// TIA Portal V17 program export: 1 tag tables, 0 data types, 1 data blocks, 5 code blocks (in call order from the OBs), 13 instance data blocks

VAR_GLOBAL   // PLC tag table "Default tag table"
   System_Byte AT %MB1 : Byte;
   FirstScan AT %M1.0 : Bool;
   DiagStatusUpdate AT %M1.1 : Bool;
   AlwaysTRUE AT %M1.2 : Bool;
   AlwaysFALSE AT %M1.3 : Bool;
   Clock_Byte AT %MB0 : Byte;
   Clock_10Hz AT %M0.0 : Bool;
   Clock_5Hz AT %M0.1 : Bool;
   "Clock_2.5Hz" AT %M0.2 : Bool;
   Clock_2Hz AT %M0.3 : Bool;
   "Clock_1.25Hz" AT %M0.4 : Bool;
   Clock_1Hz AT %M0.5 : Bool;
   "Clock_0.625Hz" AT %M0.6 : Bool;
   "Clock_0.5Hz" AT %M0.7 : Bool;
   BMS_Connect_req AT %M2.0 : Bool;
   Send_data AT %M2.2 : Bool;
   Kinco_connect_req AT %M2.1 : Bool;
   Node_ID_1 AT %MW4 : Int;
   Node_ID_2 AT %MW6 : Int;
   Connection_Established AT %M2.3 : Bool;
   Motor_1_Select_mode AT %MB3 : Byte;
   move_data_pulse AT %M2.4 : Bool;
   motor_1_control_word AT %MW10 : Word;
   LH_pulse_out AT %M2.6 : Bool;
   RH_pulse_out AT %M2.7 : Bool;
   RH_Speed AT %MD18 : DInt;
   LH_Speed AT %MD22 : DInt;
   send_data_pulse AT %M2.5 : Bool;
   node_terminate AT %I0.0 : Bool;
   motor_1_target_rpm AT %MD12 : DInt;
   motor_1_target_pos AT %MD28 : DInt;
   motor_1_profile_speed AT %MD32 : DInt;
   Tag_1 AT %I0.2 : Bool;
   wake_node_trigger AT %I0.1 : Bool;
   Motor_2_Select_mode AT %MB8 : Byte;
   motor_2_control_word AT %MW16 : Word;
   motor_2_target_rpm AT %MD36 : DInt;
   motor_2_target_pos AT %MD40 : DInt;
   motor_2_profile_speed AT %MD44 : DInt;
END_VAR

DATA_BLOCK "kinco_Data_packet_DB"   // DB9
{ S7_Optimized_Access := 'FALSE' }
VERSION : 0.1
// stored: AutoNumber true, DBAccessibleFromOPCUA true, IsOnlyStoredInLoadMemory false, IsWriteProtectedInAS false
   VAR
      Kinco_Data_Recv : Array[0..12] of Byte;
      Kinco_Data_sending_vizu : Array[0..12] of Byte;
   END_VAR
BEGIN
END_DATA_BLOCK

ORGANIZATION_BLOCK "Main"   // OB1, LAD, ProgramCycle
TITLE = "Main Program Sweep (Cycle)"
{ S7_Optimized_Access := 'TRUE' }
VERSION : 0.1
// stored: AutoNumber true, IsIECCheckEnabled false, SetENOAutomatically false
   VAR_INPUT
      Initial_Call : Bool;   // Initial call of this OB
      Remanence : Bool;   // =True, if remanent data are available
   END_VAR
BEGIN

REGION Network 1
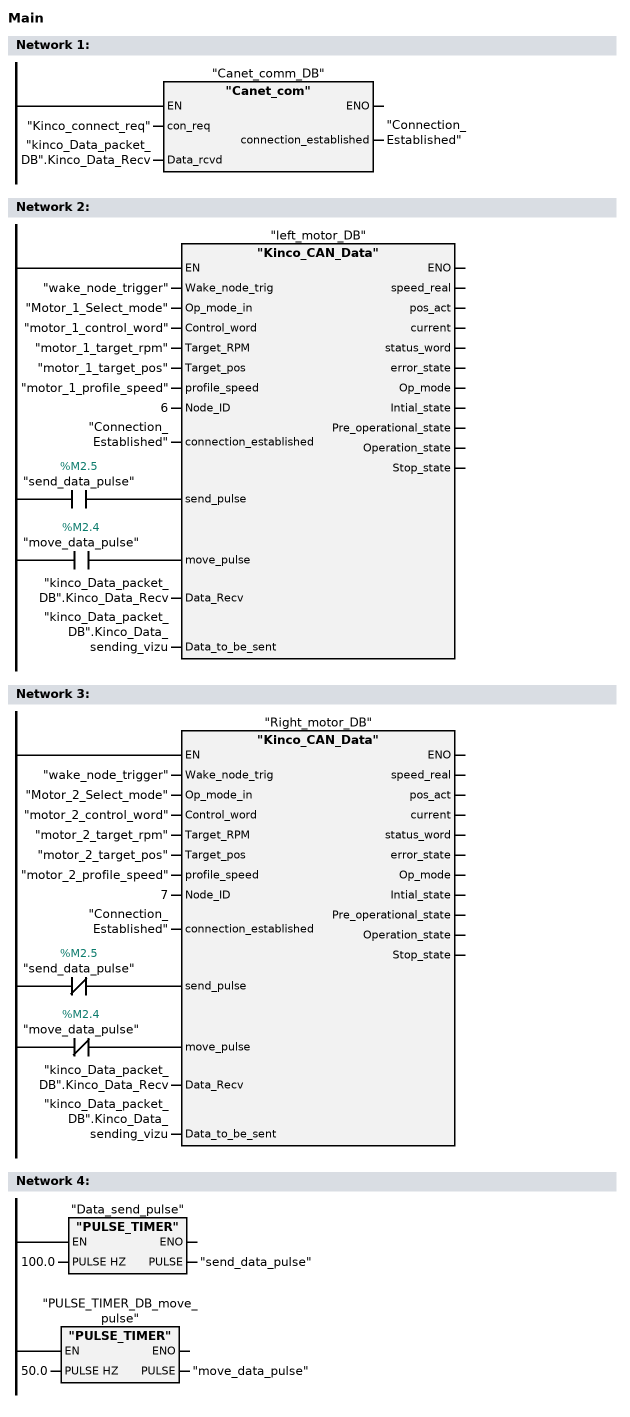
   RUNG wire#powerrail
      "Canet_comm_DB"(con_req := "Kinco_connect_req", Data_rcvd := "kinco_Data_packet_DB".Kinco_Data_Recv, connection_established => "Connection_Established")
   END_RUNG
   // the same network as SCL:
   "Canet_comm_DB"(con_req := "Kinco_connect_req",   // "Canet_com"
                   Data_rcvd := "kinco_Data_packet_DB".Kinco_Data_Recv,
                   connection_established => "Connection_Established");
END_REGION

REGION Network 2
   RUNG wire#powerrail
      "left_motor_DB"(send_pulse := wire#w1, move_pulse := wire#w2, Wake_node_trig := "wake_node_trigger", Op_mode_in := "Motor_1_Select_mode", Control_word := "motor_1_control_word", Target_RPM := "motor_1_target_rpm", Target_pos := "motor_1_target_pos", profile_speed := "motor_1_profile_speed", Node_ID := 6, connection_established := "Connection_Established", Data_Recv := "kinco_Data_packet_DB".Kinco_Data_Recv, Data_to_be_sent := "kinco_Data_packet_DB".Kinco_Data_sending_vizu, speed_real =>, pos_act =>, current =>, status_word =>, error_state =>, Op_mode =>, Intial_state =>, Pre_operational_state =>, Operation_state =>, Stop_state =>)
   END_RUNG
   RUNG wire#powerrail
      Contact( "send_data_pulse" )
   END_RUNG wire#w1
   RUNG wire#powerrail
      Contact( "move_data_pulse" )
   END_RUNG wire#w2
   // the same network as SCL:
   "left_motor_DB"(Wake_node_trig := "wake_node_trigger",   // "Kinco_CAN_Data"
                   Op_mode_in := "Motor_1_Select_mode",
                   Control_word := "motor_1_control_word",
                   Target_RPM := "motor_1_target_rpm",
                   Target_pos := "motor_1_target_pos",
                   profile_speed := "motor_1_profile_speed",
                   Node_ID := 6,
                   connection_established := "Connection_Established",
                   send_pulse := "send_data_pulse",
                   move_pulse := "move_data_pulse",
                   Data_Recv := "kinco_Data_packet_DB".Kinco_Data_Recv,
                   Data_to_be_sent := "kinco_Data_packet_DB".Kinco_Data_sending_vizu);
END_REGION

REGION Network 3
   RUNG wire#powerrail
      "Right_motor_DB"(send_pulse := wire#w1, move_pulse := wire#w2, Wake_node_trig := "wake_node_trigger", Op_mode_in := "Motor_2_Select_mode", Control_word := "motor_2_control_word", Target_RPM := "motor_2_target_rpm", Target_pos := "motor_2_target_pos", profile_speed := "motor_2_profile_speed", Node_ID := 7, connection_established := "Connection_Established", Data_Recv := "kinco_Data_packet_DB".Kinco_Data_Recv, Data_to_be_sent := "kinco_Data_packet_DB".Kinco_Data_sending_vizu, speed_real =>, pos_act =>, current =>, status_word =>, error_state =>, Op_mode =>, Intial_state =>, Pre_operational_state =>, Operation_state =>, Stop_state =>)
   END_RUNG
   RUNG wire#powerrail
      I_Contact( "send_data_pulse" )
   END_RUNG wire#w1
   RUNG wire#powerrail
      I_Contact( "move_data_pulse" )
   END_RUNG wire#w2
   // the same network as SCL:
   "Right_motor_DB"(Wake_node_trig := "wake_node_trigger",   // "Kinco_CAN_Data"
                    Op_mode_in := "Motor_2_Select_mode",
                    Control_word := "motor_2_control_word",
                    Target_RPM := "motor_2_target_rpm",
                    Target_pos := "motor_2_target_pos",
                    profile_speed := "motor_2_profile_speed",
                    Node_ID := 7,
                    connection_established := "Connection_Established",
                    send_pulse := NOT "send_data_pulse",
                    move_pulse := NOT "move_data_pulse",
                    Data_Recv := "kinco_Data_packet_DB".Kinco_Data_Recv,
                    Data_to_be_sent := "kinco_Data_packet_DB".Kinco_Data_sending_vizu);
END_REGION

REGION Network 4
   RUNG wire#powerrail
      "Data_send_pulse"("PULSE HZ" := 100.0, PULSE => "send_data_pulse")
   END_RUNG
   RUNG wire#powerrail
      "PULSE_TIMER_DB_move_pulse"("PULSE HZ" := 50.0, PULSE => "move_data_pulse")
   END_RUNG
   // the same network as SCL:
   "Data_send_pulse"("PULSE HZ" := 100.0, PULSE => "send_data_pulse");   // "PULSE_TIMER"
   "PULSE_TIMER_DB_move_pulse"("PULSE HZ" := 50.0, PULSE => "move_data_pulse");   // "PULSE_TIMER"
END_REGION
END_ORGANIZATION_BLOCK

FUNCTION_BLOCK "Canet_com"   // FB3, LAD
{ S7_Optimized_Access := 'FALSE' }
VERSION : 0.1
// stored: AutoNumber true, IsIECCheckEnabled false, SetENOAutomatically false, UDAEnableTagReadback false
   VAR_INPUT
      con_req : Bool;
   END_VAR
   VAR_OUTPUT
      connection_established : Bool;
   END_VAR
   VAR_IN_OUT
      Data_rcvd : Array[0..12] of Byte;
   END_VAR
BEGIN

REGION Network 1: Connection
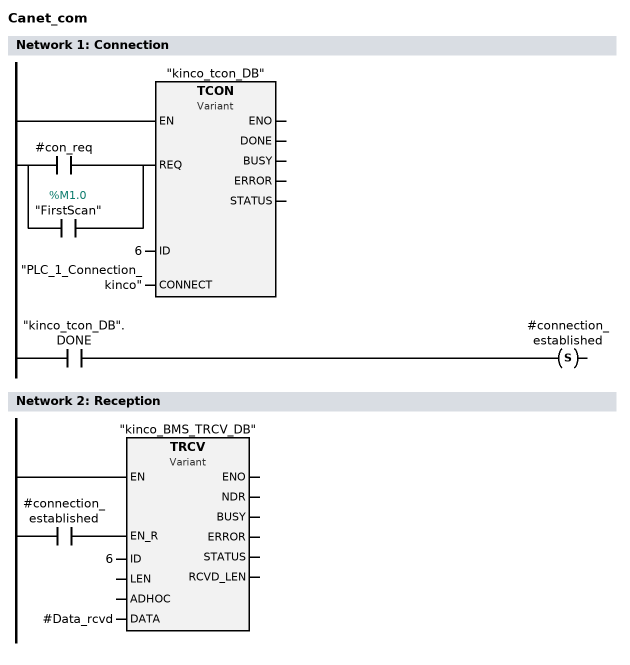
   RUNG wire#powerrail
      { S7_Templates := "[con_type := Variant, id_type := CONN_OUC]" } "kinco_tcon_DB".TCON(REQ := wire#w1, ID := 6, CONNECT := "PLC_1_Connection_kinco", DONE =>, BUSY =>, ERROR =>, STATUS =>)
   END_RUNG
   RUNG wire#powerrail
      Contact( #con_req )
   END_RUNG wire#w1
   RUNG wire#powerrail
      Contact( "FirstScan" )
   END_RUNG wire#w1
   RUNG wire#powerrail
      Contact( "kinco_tcon_DB".DONE )
      S_Coil( #connection_established )
   END_RUNG
   // the same network as SCL:
   "kinco_tcon_DB"(REQ := #con_req OR "FirstScan", ID := 6, CONNECT := "PLC_1_Connection_kinco");   // TCON
   IF "kinco_tcon_DB".DONE THEN #connection_established := TRUE; END_IF;
END_REGION

REGION Network 2: Reception
   RUNG wire#powerrail
      { S7_Templates := "[card := 1, ptr_type := Variant, value_type := UDInt, id_type := CONN_OUC]" } "kinco_BMS_TRCV_DB".TRCV(EN_R := wire#w1, ID := 6, LEN :=, ADHOC :=, DATA := #Data_rcvd, NDR =>, BUSY =>, ERROR =>, STATUS =>, RCVD_LEN =>)
   END_RUNG
   RUNG wire#powerrail
      Contact( #connection_established )
   END_RUNG wire#w1
   // the same network as SCL:
   "kinco_BMS_TRCV_DB"(EN_R := #connection_established, ID := 6, DATA := #Data_rcvd);   // TRCV
END_REGION
END_FUNCTION_BLOCK

FUNCTION_BLOCK "Kinco_CAN_Data"   // FB4, LAD
{ S7_Optimized_Access := 'TRUE' }
VERSION : 0.1
// stored: AutoNumber true, IsIECCheckEnabled false, IsRetainMemResEnabled false, MemoryReserve 100, SetENOAutomatically false, UDAEnableTagReadback false
   VAR_INPUT
      Wake_node_trig : Bool;
      Op_mode_in : Byte;
      Control_word : Word;
      Target_RPM : DInt;
      Target_pos : DInt;
      profile_speed : DInt;
      Node_ID : Int;
      connection_established : Bool;
      send_pulse : Bool;
      move_pulse : Bool;
      Data_Recv { ExternalAccessible := 'False'; ExternalVisible := 'False'; ExternalWritable := 'False'} : Array[0..12] of Byte;
   END_VAR
   VAR_OUTPUT
      speed_real : DInt;
      pos_act : DInt;
      current : Real;
      status_word : Word;
      error_state : Word;
      Op_mode : Byte;
      Intial_state : Bool;
      Pre_operational_state : Bool;
      Operation_state : Bool;
      Stop_state : Bool;
   END_VAR
   VAR_IN_OUT
      Data_to_be_sent : Array[0..12] of Byte;
   END_VAR
   VAR
      tsend_inst : TSEND;
      Target_RPM_hex { S7_SetPoint := 'True'} : DWord;
      Target_pos_hex : DWord;
      profile_speed_hex : DWord;
   END_VAR
BEGIN

REGION Network 1: Data_sending
   // Send_data_at_100HZ
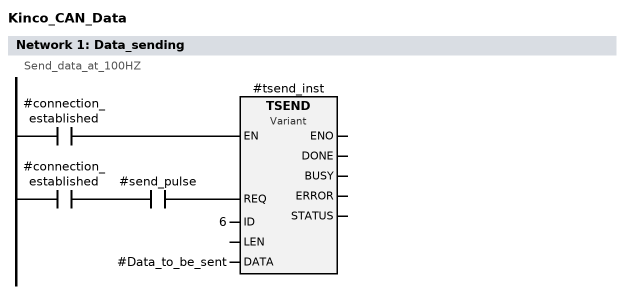
   RUNG wire#powerrail
      Contact( #connection_established )
      { S7_Templates := "[data_type := Variant, len_type := UDInt, id_type := CONN_OUC]" } #tsend_inst.TSEND(REQ := wire#w1, ID := 6, LEN :=, DATA := #Data_to_be_sent, DONE =>, BUSY =>, ERROR =>, STATUS =>)
   END_RUNG
   RUNG wire#powerrail
      Contact( #connection_established )
      Contact( #send_pulse )
   END_RUNG wire#w1
   // the same network as SCL:
   IF #connection_established THEN
       #tsend_inst(REQ := #connection_established AND #send_pulse, ID := 6, DATA := #Data_to_be_sent);   // TSEND
   END_IF;
END_REGION

REGION Network 2 (SCL): Data_parsing
   IF #Data_Recv[3]= 16#01 AND (#Data_Recv[4]= 16#80 + #Node_ID) THEN
       #speed_real := DWORD_TO_DINT(SWAP(%DB9.))/2730.66;
       #pos_act := DWORD_TO_DINT(SWAP(%DB9.));
   END_IF;

   IF %DB9. = (16#0280 + #Node_ID) THEN
       #current := INT_TO_REAL(SWAP(%DB9.)) / 36.20;
       #Op_mode := %DB9.;
   END_IF;

   IF %DB9. = (16#0380 + #Node_ID) THEN
       #status_word := SWAP(%DB9.);
       #error_state := SWAP(%DB9.);
   END_IF;
END_REGION

REGION Network 3 (SCL): wake_node
   IF "Connection_Established" AND (#status_word = 16#0000 OR #Wake_node_trig) AND #move_pulse THEN
       #Data_to_be_sent[3] := 16#00;
       #Data_to_be_sent[4] := 16#00;
       #Data_to_be_sent[5] := 16#01;
       #Data_to_be_sent[6] := #Node_ID;
       #Data_to_be_sent[7] := 16#00;
       #Data_to_be_sent[8] := 16#00;
       #Data_to_be_sent[9] := 16#00;
       #Data_to_be_sent[10] := 16#00;
       #Data_to_be_sent[11] := 16#00;
       #Data_to_be_sent[12] := 16#00;
   END_IF;
END_REGION

REGION Network 4 (SCL): State_definition
   IF #status_word.%X0 = 1 AND #status_word.%X1 = 0 AND #status_word.%X2 = 0 AND #status_word.%X3 = 0 AND #status_word.%X14 = 0 THEN
       #Intial_state := TRUE;
       #Pre_operational_state := FALSE;
       #Operation_state := FALSE;
       #Stop_state := FALSE;
   ELSIF #status_word.%X0 = 1 AND #status_word.%X1 = 0 AND #status_word.%X2 = 0 AND #status_word.%X3 = 0 AND #status_word.%X14 = 1 THEN
       #Intial_state := FALSE;
       #Pre_operational_state := TRUE;
       #Operation_state := FALSE;
       #Stop_state := FALSE;
   ELSIF #status_word.%X0 = 1 AND #status_word.%X1 = 1 AND #status_word.%X2 = 1 AND #status_word.%X3 = 0 AND #status_word.%X14 = 1 THEN
       #Intial_state := FALSE;
       #Pre_operational_state := FALSE;
       #Operation_state := TRUE;
       #Stop_state := FALSE;
   ELSIF #status_word.%X0 = 1 AND #status_word.%X1 = 0 AND #status_word.%X2 = 0 AND #status_word.%X3 = 0 AND #status_word.%X14 = 1 THEN
       #Intial_state := FALSE;
       #Pre_operational_state := FALSE;
       #Operation_state := FALSE;
       #Stop_state := TRUE;
   END_IF;
END_REGION

REGION Network 5 (SCL): Conditions_n_data_assignment
   #Target_RPM_hex := DINT_TO_DWORD(#Target_RPM * 2731);
   #Target_pos_hex := DINT_TO_DWORD(#Target_pos);
   #profile_speed_hex := DINT_TO_DWORD(#profile_speed * 2731);
   IF #Stop_state THEN
       #Control_word := 16#0086;
   END_IF;
   IF #Op_mode_in <> #Op_mode AND NOT(#Stop_state) THEN
       #Control_word := 16#0006;
   END_IF;
END_REGION

REGION Network 6 (SCL): Standard_packet
   // Move data at 10 hz
   #Data_to_be_sent[0] := 16#08;
   #Data_to_be_sent[1] := 16#00;
   #Data_to_be_sent[2] := 16#00;
   IF (#Pre_operational_state OR #Intial_state OR #Stop_state OR #Op_mode_in <> #Op_mode OR (#Control_word=16#0006 OR #Control_word=16#0086)) AND NOT(#Wake_node_trig) AND #move_pulse THEN
       #Data_to_be_sent[3] := 16#02;
       #Data_to_be_sent[4] := #Node_ID;
       #Data_to_be_sent[5] := #Control_word.%B0;
       #Data_to_be_sent[6] := #Control_word.%B1;
       #Data_to_be_sent[7] := #Op_mode_in;
       #Data_to_be_sent[8] := 16#00;
       #Data_to_be_sent[9] := 16#00;
       #Data_to_be_sent[10] := 16#00;
       #Data_to_be_sent[11] := 16#00;
       #Data_to_be_sent[12] := 16#00;
   END_IF;
   IF #Operation_state AND NOT (#Pre_operational_state OR #Intial_state OR #Stop_state) AND (#Op_mode_in = 16#03) AND NOT(#Control_word=16#0006 OR #Control_word=16#0086) AND #Op_mode_in=#Op_mode AND NOT(#Wake_node_trig) AND #move_pulse THEN
       #Data_to_be_sent[3] := 16#03;
       #Data_to_be_sent[4] := #Node_ID;
       #Data_to_be_sent[5] := #Target_RPM_hex.%B0;
       #Data_to_be_sent[6] := #Target_RPM_hex.%B1;
       #Data_to_be_sent[7] := #Target_RPM_hex.%B2;
       #Data_to_be_sent[8] := #Target_RPM_hex.%B3;
       #Data_to_be_sent[9] := 16#00;
       #Data_to_be_sent[10] := 16#00;
       #Data_to_be_sent[11] := 16#00;
       #Data_to_be_sent[12] := 16#00;
   END_IF;
   IF #Operation_state AND NOT(#Pre_operational_state OR #Intial_state OR #Stop_state) AND (#Op_mode_in = 16#01) AND NOT(#Control_word=16#0006 OR #Control_word=16#0086) AND #Op_mode_in=#Op_mode AND NOT(#Wake_node_trig) AND #move_pulse THEN
       #Data_to_be_sent[3] := 16#04;
       #Data_to_be_sent[4] := #Node_ID;
       #Data_to_be_sent[5] := #profile_speed_hex.%B0;
       #Data_to_be_sent[6] := #profile_speed_hex.%B1;
       #Data_to_be_sent[7] := #profile_speed_hex.%B2;
       #Data_to_be_sent[8] := #profile_speed_hex. %B3;
       #Data_to_be_sent[9] := #Target_pos_hex.%B0;
       #Data_to_be_sent[10] := #Target_pos_hex.%B1;
       #Data_to_be_sent[11] := #Target_pos_hex.%B2;
       #Data_to_be_sent[12] := #Target_pos_hex.%B3;
   END_IF;
END_REGION
END_FUNCTION_BLOCK

FUNCTION_BLOCK "PULSE_TIMER"   // FB5, LAD
{ S7_Optimized_Access := 'TRUE' }
VERSION : 0.1
// stored: AutoNumber true, IsIECCheckEnabled false, IsRetainMemResEnabled false, MemoryReserve 100, SetENOAutomatically false, UDAEnableTagReadback false
   VAR_INPUT
      "PULSE HZ" : Real;
   END_VAR
   VAR_OUTPUT
      PULSE : Bool;
   END_VAR
   VAR
      Clock_Timer_1 : IEC_TIMER;
      Clock_Timer_2 : IEC_TIMER;
      "Time(s)" { S7_SetPoint := 'True'} : Real;
      "Time(ms)" : Real;
      "Time" : Int;
   END_VAR
BEGIN

REGION Network 1: Timer Loop
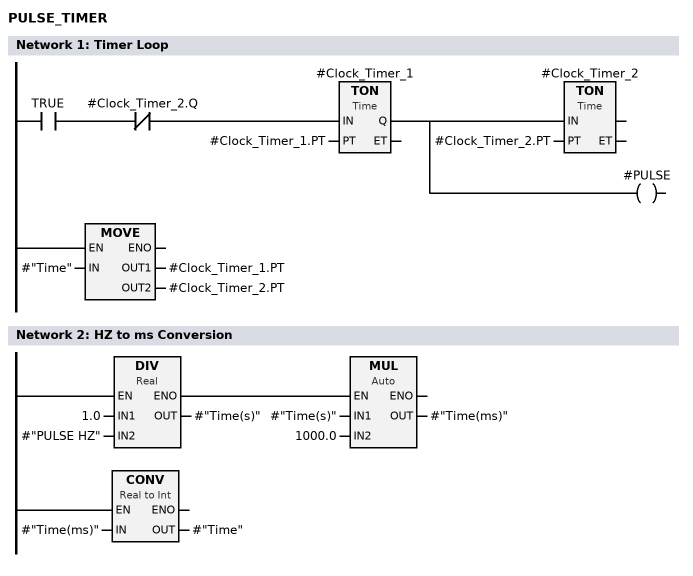
   RUNG wire#powerrail
      Contact( TRUE )
      I_Contact( #Clock_Timer_2.Q )
      { S7_Templates := "time_type := Time" } #Clock_Timer_1.TON(pt := #Clock_Timer_1.PT, et =>)
      wire#w1
      { S7_Templates := "time_type := Time" } #Clock_Timer_2.TON(pt := #Clock_Timer_2.PT, et =>)
   END_RUNG
   RUNG wire#w1
      Coil( #PULSE )
   END_RUNG
   RUNG wire#powerrail
      Move(in := #"Time", out1 => #Clock_Timer_1.PT, out2 => #Clock_Timer_2.PT)
   END_RUNG
   // the same network as SCL:
   #Clock_Timer_1.TON(IN := TRUE AND NOT #Clock_Timer_2.Q, PT := #Clock_Timer_1.PT);
   #Clock_Timer_2.TON(IN := #Clock_Timer_1.Q, PT := #Clock_Timer_2.PT);
   #PULSE := #Clock_Timer_1.Q;
   #Clock_Timer_1.PT := #"Time";
   #Clock_Timer_2.PT := #"Time";
END_REGION

REGION Network 2: HZ to ms Conversion
   RUNG wire#powerrail
      { S7_Templates := "SrcType := Real" } Div(in1 := 1.0, in2 := #"PULSE HZ", out => #"Time(s)")
      Mul(in1 := #"Time(s)", in2 := 1000.0, out => #"Time(ms)")
   END_RUNG
   RUNG wire#powerrail
      { S7_Templates := "[SrcType := Real, DestType := Int]" } Convert(in := #"Time(ms)", out => #"Time")
   END_RUNG
   // the same network as SCL:
   #"Time(s)" := 1.0 / #"PULSE HZ";
   #"Time(ms)" := #"Time(s)" * 1000.0;
   #"Time" := REAL_TO_INT(#"Time(ms)");
END_REGION
END_FUNCTION_BLOCK

FUNCTION_BLOCK "Main_Safety_RTG1"   // FB1, F_FBD
{ S7_Optimized_Access := 'TRUE' }
VERSION : 0.1
// stored: AutoNumber false, IsIECCheckEnabled false, UDAEnableTagReadback false
BEGIN
END_FUNCTION_BLOCK

DATA_BLOCK "Canet_comm_DB"   // DB5
VERSION : 0.1
// stored: AutoNumber true, DBAccessibleFromOPCUA true, InstanceOfName Canet_com, InstanceOfType FB
"Canet_com"
BEGIN
END_DATA_BLOCK

DATA_BLOCK "Data_move_pulse"   // DB3
VERSION : 0.1
// stored: AutoNumber true, DBAccessibleFromOPCUA true, InstanceOfName PULSE_TIMER, InstanceOfType FB
"PULSE_TIMER"
BEGIN
END_DATA_BLOCK

DATA_BLOCK "Data_send_pulse"   // DB13
VERSION : 0.1
// stored: AutoNumber true, DBAccessibleFromOPCUA true, InstanceOfName PULSE_TIMER, InstanceOfType FB
"PULSE_TIMER"
BEGIN
END_DATA_BLOCK

DATA_BLOCK "Main_Safety_RTG1_DB"   // DB1, F_DB
NAME : FUSI
VERSION : 0.1
// stored: AutoNumber true, DBAccessibleFromOPCUA true, InstanceOfName Main_Safety_RTG1, InstanceOfType FB
"Main_Safety_RTG1"
BEGIN
END_DATA_BLOCK

DATA_BLOCK "PULSE_TIMER_DB"   // DB16
VERSION : 0.1
// stored: AutoNumber true, DBAccessibleFromOPCUA true, InstanceOfName PULSE_TIMER, InstanceOfType FB
"PULSE_TIMER"
BEGIN
END_DATA_BLOCK

DATA_BLOCK "PULSE_TIMER_DB_move_pulse"   // DB2
VERSION : 0.1
// stored: AutoNumber true, DBAccessibleFromOPCUA true, InstanceOfName PULSE_TIMER, InstanceOfType FB
"PULSE_TIMER"
BEGIN
END_DATA_BLOCK

DATA_BLOCK "Right_motor_DB"   // DB10
VERSION : 0.1
// stored: AutoNumber true, DBAccessibleFromOPCUA true, InstanceOfName Kinco_CAN_Data, InstanceOfType FB
"Kinco_CAN_Data"
BEGIN
END_DATA_BLOCK

DATA_BLOCK "left_motor_DB"   // DB6
VERSION : 0.1
// stored: AutoNumber true, DBAccessibleFromOPCUA true, InstanceOfName Kinco_CAN_Data, InstanceOfType FB
"Kinco_CAN_Data"
BEGIN
END_DATA_BLOCK

DATA_BLOCK "Canet_com_DB"   // DB20
VERSION : 0.1
// stored: AutoNumber true, DBAccessibleFromOPCUA true, InstanceOfName Canet_com, InstanceOfType FB
"Canet_com"
BEGIN
END_DATA_BLOCK

DATA_BLOCK "Kinco_CAN_Data_DB"   // DB18
VERSION : 0.1
// stored: AutoNumber true, DBAccessibleFromOPCUA true, InstanceOfName Kinco_CAN_Data, InstanceOfType FB
"Kinco_CAN_Data"
BEGIN
END_DATA_BLOCK

DATA_BLOCK "PLC_1_Connection_kinco"   // DB11
{ S7_Optimized_Access := 'TRUE' }
// stored: AutoNumber true, DBAccessibleFromOPCUA true, InstanceOfName TCON_IP_v4, OfSystemLibElement TCON_IP_v4, OfSystemLibVersion 1.0
"TCON_IP_v4"
   // VAR
   //    InterfaceId : HW_ANY := 64;
   //    ID : CONN_OUC := 6;
   //    ConnectionType : Byte;
   //    ActiveEstablished : Bool := true;
   //    RemoteAddress { S7_SetPoint := 'True'} : IP_V4;
   //    RemotePort : UInt := 2005;
   //    LocalPort : UInt := 0;
   // END_VAR
BEGIN
   RemoteAddress.ADDR[1] := 192;
   RemoteAddress.ADDR[2] := 168;
   RemoteAddress.ADDR[3] := 1;
   RemoteAddress.ADDR[4] := 199;
END_DATA_BLOCK

DATA_BLOCK "kinco_BMS_TRCV_DB"   // DB8
// stored: AutoNumber true, DBAccessibleFromOPCUA true, InstanceOfName TRCV, OfSystemLibElement TRCV, OfSystemLibVersion 4.0
"TRCV"
   // VAR_INPUT
   //    EN_R : Bool;
   //    ID : CONN_OUC;
   //    LEN : UDInt;
   //    ADHOC : Bool;
   // END_VAR
   // VAR_OUTPUT
   //    NDR : Bool;
   //    BUSY : Bool;
   //    ERROR : Bool;
   //    STATUS : Word;
   //    RCVD_LEN : UDInt;
   // END_VAR
   // VAR_IN_OUT
   //    DATA : Variant;
   //    ADDR : Variant;
   // END_VAR
BEGIN
END_DATA_BLOCK

DATA_BLOCK "kinco_tcon_DB"   // DB7
// stored: AutoNumber true, DBAccessibleFromOPCUA true, InstanceOfName TCON, OfSystemLibElement TCON, OfSystemLibVersion 4.0
"TCON"
   // VAR_INPUT
   //    REQ : Bool;
   //    ID : CONN_OUC;
   // END_VAR
   // VAR_OUTPUT
   //    DONE : Bool;
   //    BUSY : Bool;
   //    ERROR : Bool;
   //    STATUS : Word;
   // END_VAR
   // VAR_IN_OUT
   //    CONNECT : Variant;
   // END_VAR
BEGIN
END_DATA_BLOCK
